// TIA Portal V19 export
TYPE "LEXCHANGETRAY_typePlasticEm5_deliver_interface"
// stored: Access Published
   STRUCT
      init : Bool;
      roller : "LEXCHANGETRAY_typePlasticEm5_toRollerDeliver";
      handlingXyz { S7_SetPoint := 'True'} : "LEXCHANGETRAY_typePlasticEm5_toHandlingXyzDeliver";
   END_STRUCT;
END_TYPE
